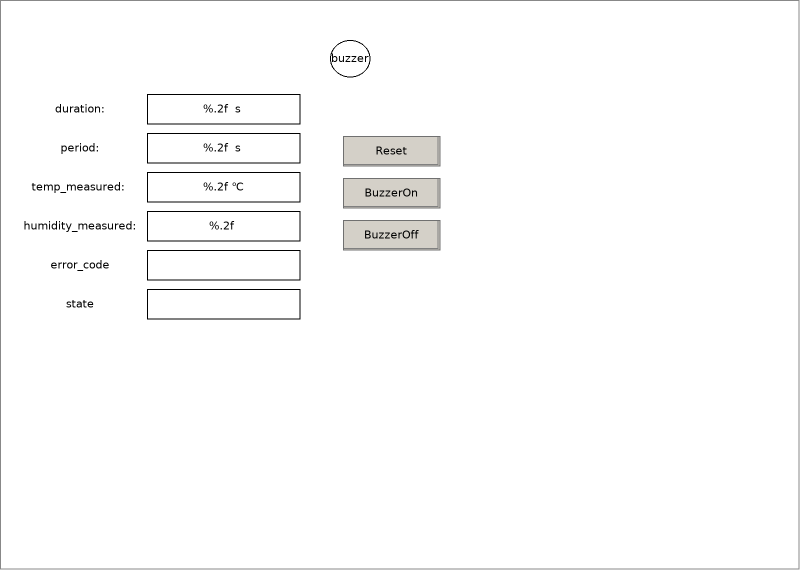
VISUALIZATION VIS_SystemEnvironment  // 800x570
    Button (343,178 97x30), "BuzzerOn", colour toggle: GVL_API.stSystemEnvironment.BuzzerOn
        toggle GVL_API.stSystemEnvironment.BuzzerOn
    Button (343,136 97x30), "Reset", colour toggle: GVL_API.stSystemEnvironment.Reset
        toggle GVL_API.stSystemEnvironment.Reset
    Button (343,220 97x30), "BuzzerOff", colour toggle: GVL_API.stSystemEnvironment.BuzzerOff
        toggle GVL_API.stSystemEnvironment.BuzzerOff
    Ellipse (330,40 40x37), "buzzer", colour toggle: stOutput.bqBuzzer
    Rectangle (147,94 153x30), "%.2f s", text variable: GVL_API.stSystemEnvironment.duration
        OnMouseDown: write GVL_API.stSystemEnvironment.duration via Default
    Rectangle (147,133 153x30), "%.2f s", text variable: GVL_API.stSystemEnvironment.period
        OnMouseDown: write GVL_API.stSystemEnvironment.period via Default
    Rectangle (147,211 153x30), "%.2f", text variable: GVL_API.stSystemEnvironment.humidity_measured
        OnMouseDown: write GVL_API.stRoolToRool[1].acceleration via Default
    Rectangle (147,172 153x30), "%.2f ℃", text variable: GVL_API.stSystemEnvironment.temp_measured
    Rectangle (147,250 153x30), text list: 'TextList_EnvironmentError', text index: GVL_API.stSystemEnvironment.error_code
    Rectangle (147,289 153x30), text list: 'TextList_EnvironmentState', text index: GVL_API.stSystemEnvironment.state
    Label (15,250 130x30), "error_code"
    Label (15,289 130x30), "state"
    Label (15,211 130x30), "humidity_measured:"
    Label (15,172 130x30), "temp_measured:"
    Label (15,133 130x30), "period:"
    Label (15,94 130x30), "duration:"
END_VISUALIZATION

(* stored: Version 1.1.0.1, ProductVersion 3.1.4024.11
   Visu VIS_SystemEnvironment: Id {3bcbff76-95a0-46df-a04d-eefcc56596cc} *)
